Fanuc KAREL source: ka00077.KL

-- PROVISIONAL review KL for V1013-1; original PC SHA256 09c007bfb16404d18265effcc1c26d6f34386f0cea27e71f2e9dcfc7410e7d6f
-- Incomplete behavior may be omitted. Consult companion uncertainty JSON. Do not deploy.
PROGRAM KA00077
%NOLOCKGROUP
-- UNRESOLVED_DECL SRC type=000106
-- UNRESOLVED_DECL DST type=000101
BEGIN
  -- UNRESOLVED_PC offsets 5-20; opcodes 2E,22,32,35
  -- UNRESOLVED_PC offsets 25-45; opcodes 49,7E,4A
  -- UNRESOLVED_PC offsets 50-54; opcodes 7F
END KA00077
